TYPE
    ST_WaitSyncManager : STRUCT
        ID         : E_WaitSync;
        Active     : BOOL;
        AreaNeeded : ARRAY[1..30] OF BOOL;
        State      : UDINT;
    END_STRUCT
END_TYPE

(* stored: Version 1.1.0.1
   DUT ST_WaitSyncManager: Id {a6e2ed3d-2491-4b0a-b64d-c2ffdf027c8f} *)
